TYPE ST_InputsTransferCC :
(**************************************************************************************
 * 	Application		:	BoxControl Framework
 *	Revision		:	$Revision: 417092 $
 *	Revision date	:	$Date: 2018-11-14 12:58:58 +0100 (Mi., 14 Nov 2018) $
 *	Last changed by	:	$Author: q8aberh $
 *	URL				:	$URL: http://almscdc.swisslog.com/repo/SWPD/Development/ProMove/02_Controls/ProBox/03_Implementation/01_DevelopmentProject/01_Software/ProBox_COE/ProBox_DevProj_v1.0/PLC_1/20_Product/10_App/12_E_Functions/11_ProBox/21_LowLiftUnit/10_App/01_DUTs/ST_Input $
 *
 *	Purpose			:	Function specific inputs.
 *
 * ------------------------------------------------------------------------------------
 *	Copyright Swisslog [IP AG], Switzerland. All rights reserved.
 * 
 * ------------------------------------------------------------------------------------
 *	
 * 	Revision History: 
 *
 * 	VERSION			DATE			INITIALS			DESCRIPTION
 *	0.1				01.01.2001		swl					Example
 *
 **************************************************************************************)	
STRUCT
	Sensor_Stop_12			: BOOL; // Sensor stop axis 1-2 forward
	Sensor_Slow_12			: BOOL; // Sensor slow speed axis 1-2 forward
	Sensor_Creep_12			: BOOL; // Sensor creep speed axis 1-2 forward
	Sensor_Overhang_12		: BOOL; // Sensor overhang axis 1-2 forward	
	Sensor_Stop_21			: BOOL; // Sensor stop axis 1-2 reverse
	Sensor_Slow_21			: BOOL; // Sensor slow speed axis 1-2 reverse
	Sensor_Creep_21			: BOOL; // Sensor creep speed axis 1-2 reverse
	Sensor_Overhang_21		: BOOL; // Sensor overhang axis 1-2 reverse	
	Sensor_Pos_Left			: BOOL; // Sensor position left    
	Sensor_Creep_Left		: BOOL; // Sensor creep speed left 
	Sensor_EndLimit_Left	: BOOL; // Sensor end limit left	  
	Sensor_Pos_Right		: BOOL; // Sensor position right   
	Sensor_Creep_Right		: BOOL; // Sensor creep speed right
	Sensor_EndLimit_Right	: BOOL; // Sensor end limit right  
	Signal_MotorUnitOK		: BOOL; // Signal motor unit OK	   
END_STRUCT
END_TYPE

(* stored: Version 1.1.0.1, ProductVersion 3.1.4022.12
   DUT ST_InputsTransferCC: Id {7c2d4fdd-ede4-4937-bb56-ce4e94b67cc0} *)
